// TIA Portal V19 export
FUNCTION_BLOCK "TYPIC_C401_IF_RSS"   // FB106, FBD
TITLE = TYPIC_C401_IF_RSS: RSS-bord
{ S7_Optimized_Access := 'TRUE' }
AUTHOR : OCOTECH
FAMILY : Typical
NAME : C401.701
// Logisch Object Besturing: C401.701
// 
// De interne functie RSSobord verzorgt de bewaking van een RSSobord en stuurt de informatie door naar de subfunctie.
// stored: MemoryReserve 10, SetENOAutomatically false
   VAR_INPUT
      EXT_AUT { ExternalAccessible := 'False'; ExternalVisible := 'False'; ExternalWritable := 'False'} : Bool;   // Externe (hoofd) beveiliging (1 = OK)
      EXT_HW { ExternalAccessible := 'False'; ExternalVisible := 'False'; ExternalWritable := 'False'} : Bool;   // Sturings hardware (PLC) bewaking (1 = OK)
      IN_STO_NOK { ExternalAccessible := 'False'; ExternalVisible := 'False'; ExternalWritable := 'False'} : Bool;   // Storing aanwezig die niet observeerbaar tot gevolg heeft
      IN_STO_OK { ExternalAccessible := 'False'; ExternalVisible := 'False'; ExternalWritable := 'False'} : Bool;   // Storing aanwezig die observeerbaarheid niet beinvloed
      IN_LUS_STO { ExternalAccessible := 'False'; ExternalVisible := 'False'; ExternalWritable := 'False'} : Bool;   // Storing van het luspaar
      IN_STS { ExternalAccessible := 'False'; ExternalVisible := 'False'; ExternalWritable := 'False'} : String[8];   // Naam van de getoonde beeldstand (bitmap) op het bord
      IN_PRTG_STO { ExternalAccessible := 'False'; ExternalVisible := 'False'; ExternalWritable := 'False'} : Bool;   // Storingsmelding RSS-bord vanuit PRTG
      IN_AUT_C401 { ExternalAccessible := 'False'; ExternalVisible := 'False'; ExternalWritable := 'False'} : Bool;   // Beveiligingen: serie geschakelde terugmelding (1 = OK)
   END_VAR
   VAR_OUTPUT
      VAR_IF_RSS { ExternalAccessible := 'False'; ExternalVisible := 'False'; ExternalWritable := 'False'} : "C401_VAR_IF_RSS_TYPIC";   // Struct met alle variabelen naar bovenliggende functies
   END_VAR
   VAR
      STO { ExternalWritable := 'False'} : Struct   // Storingen
         A001 { ExternalAccessible := 'False'; ExternalVisible := 'False'} : Bool;   // Beveiliging aangesproken
         A002 { ExternalAccessible := 'False'; ExternalVisible := 'False'} : Bool;   // Storing luspaar
         A003 { ExternalAccessible := 'False'; ExternalVisible := 'False'} : Bool;   // Storing RSS-bord gedetecteerd door PRTG
         A004 { ExternalAccessible := 'False'; ExternalVisible := 'False'} : Bool;   // Storing RSS-bord
         A005 { ExternalAccessible := 'False'; ExternalVisible := 'False'} : Bool;   // Algemene storing RSS-bord
      END_STRUCT;
      VAR { ExternalWritable := 'False'} : Struct   // Variabelen
         STS { ExternalAccessible := 'False'; ExternalVisible := 'False'} : String[8];   // Naam van de getoonde beeldstand (bitmap) op het bord
         EXT_AUT { ExternalAccessible := 'False'; ExternalVisible := 'False'} : Bool;   // Externe (hoofd) beveiliging aangesproken
         EXT_HW { ExternalAccessible := 'False'; ExternalVisible := 'False'} : Bool;   // Sturings hardware (PLC) in storing
      END_STRUCT;
   END_VAR
BEGIN

REGION Network 1: START
END_REGION

REGION Network 2: +++ Storingen +++
   // Verzamelen storingsmeldingen.
END_REGION

REGION Network 3: Storing A001: Beveiliging aangesproken
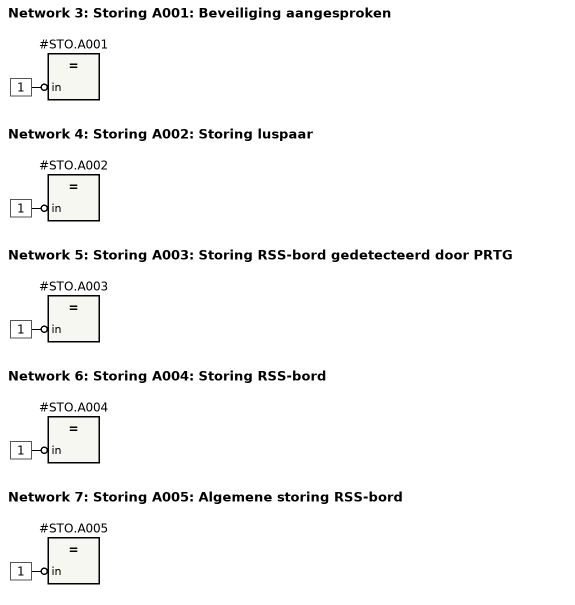
   #STO.A001 := NOT 1;
END_REGION

REGION Network 4: Storing A002: Storing luspaar
   #STO.A002 := NOT 1;
END_REGION

REGION Network 5: Storing A003: Storing RSS-bord gedetecteerd door PRTG
   #STO.A003 := NOT 1;
END_REGION

REGION Network 6: Storing A004: Storing RSS-bord
   #STO.A004 := NOT 1;
END_REGION

REGION Network 7: Storing A005: Algemene storing RSS-bord
   #STO.A005 := NOT 1;
END_REGION

REGION Network 8: +++ Beeldstand +++
   // Doorgeven van de status van het RSS-bord naar de subfunctie.
END_REGION

REGION Network 9 (SCL): EINDE
   // Variabelen van intern scada rakvlak naar outputs copieren
   #VAR_IF_RSS.STS := #VAR.STS;
   #VAR_IF_RSS.EXT_AUT := #VAR.EXT_AUT;
   #VAR_IF_RSS.EXT_HW := #VAR.EXT_HW;
   #VAR_IF_RSS.STO := #STO;
END_REGION
END_FUNCTION_BLOCK
